% RSLogix 500 project I2P JOB 7 Brandon F.RSS, saved by version 10.00.00.00 %
PROJECT "ML05B"    % processor: Bul.1763 MicroLogix 1100 Series B %

PROGRAM FILES
  LAD 2   2 rungs

DATA FILES
  O0 OUTPUT  4 elements
  I1 INPUT  6 elements
  S2 STATUS  66 elements
  B3 BINARY  1 elements
  T4 TIMER  1 elements
  C5 COUNTER  1 elements
  R6 CONTROL  1 elements
  N7 INTEGER  1 elements
  F8 FLOAT  1 elements

LADDER 2
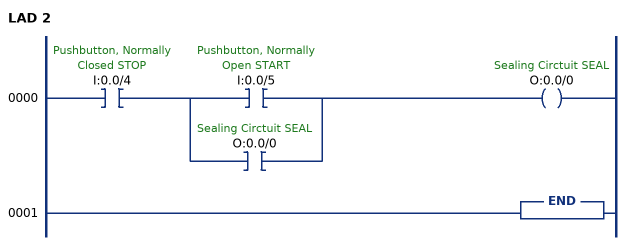
% Rung: 0 %  % edit flag set %
SOR XIC I:0.0/4 BST XIC I:0.0/5 NXB XIC O:0.0/0 BND OTE O:0.0/0 EOR
%   I:0.0/4  STOP  "Pushbutton, Normally Closed" %
%   I:0.0/5  START  "Pushbutton, Normally Open" %
%   O:0.0/0  SEAL  "Sealing Circtuit" %
% Rung: 1 %
SOR END EOR
